% RSLogix 500 project Digital_Filling_Station.RSS, saved by version 8.30.00.16 %
PROJECT "P2"    % processor: Bul.1763 MicroLogix 1100 Series B %

PROGRAM FILES
  LAD 2   4 rungs
  LAD 3 "IO"  8 rungs
  LAD 4 "CONTROL"  6 rungs
  LAD 5 "CYCLE"  5 rungs

DATA FILES
  O0 OUTPUT  4 elements
  I1 INPUT  6 elements
  S2 STATUS  66 elements
  B3 BINARY  1 elements
  T4 TIMER  1 elements
  C5 COUNTER  1 elements
  R6 CONTROL  1 elements
  N7 INTEGER  1 elements
  F8 FLOAT  1 elements

LADDER 2
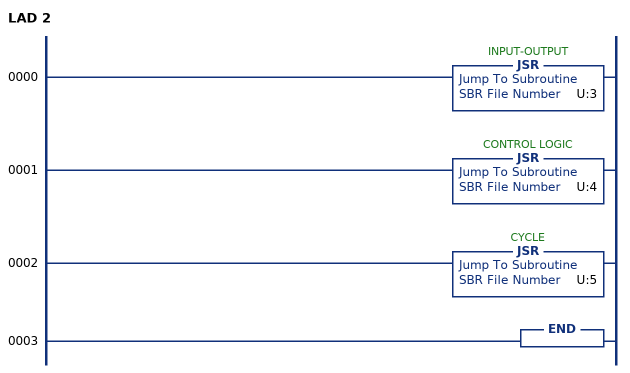
% Rung: 0 %
SOR JSR U:3 EOR
%   U:3  "INPUT-OUTPUT" %
% Rung: 1 %
SOR JSR U:4 EOR
%   U:4  "CONTROL LOGIC" %
% Rung: 2 %
SOR JSR U:5 EOR
%   U:5  "CYCLE" %
% Rung: 3 %
SOR END EOR

LADDER 3 "IO"
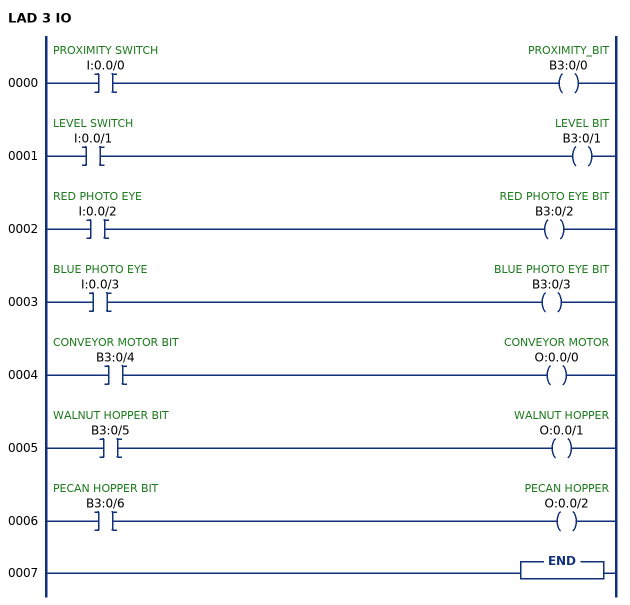
% Rung: 0 %
SOR XIC I:0.0/0 OTE B3:0/0 EOR
%   I:0.0/0  "PROXIMITY SWITCH" %
%   B3:0/0  "PROXIMITY_BIT" %
% Rung: 1 %
SOR XIC I:0.0/1 OTE B3:0/1 EOR
%   I:0.0/1  "LEVEL SWITCH" %
%   B3:0/1  "LEVEL BIT" %
% Rung: 2 %
SOR XIC I:0.0/2 OTE B3:0/2 EOR
%   I:0.0/2  "RED PHOTO EYE" %
%   B3:0/2  "RED PHOTO EYE BIT" %
% Rung: 3 %
SOR XIC I:0.0/3 OTE B3:0/3 EOR
%   I:0.0/3  "BLUE PHOTO EYE" %
%   B3:0/3  "BLUE PHOTO EYE BIT" %
% Rung: 4 %
SOR XIC B3:0/4 OTE O:0.0/0 EOR
%   B3:0/4  "CONVEYOR MOTOR BIT" %
%   O:0.0/0  "CONVEYOR MOTOR" %
% Rung: 5 %
SOR XIC B3:0/5 OTE O:0.0/1 EOR
%   B3:0/5  "WALNUT HOPPER BIT" %
%   O:0.0/1  "WALNUT HOPPER" %
% Rung: 6 %
SOR XIC B3:0/6 OTE O:0.0/2 EOR
%   B3:0/6  "PECAN HOPPER BIT" %
%   O:0.0/2  "PECAN HOPPER" %
% Rung: 7 %
SOR END EOR

LADDER 4 "CONTROL"
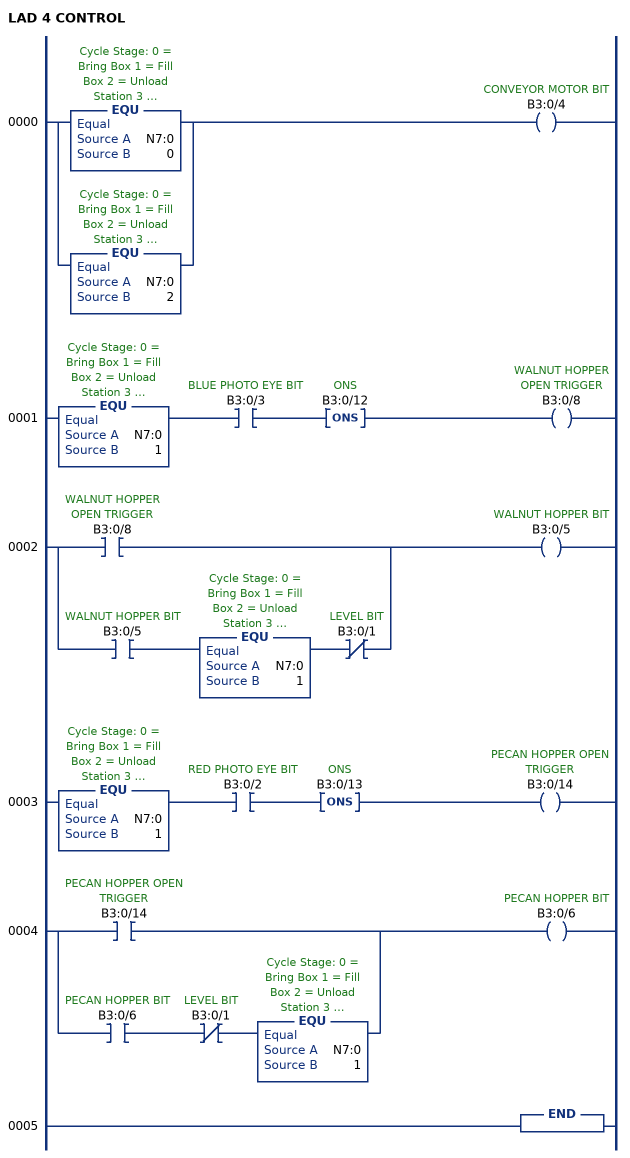
% Rung: 0 %
SOR BST EQU N7:0 0 NXB EQU N7:0 2 BND OTE B3:0/4 EOR
%   N7:0  "Cycle Stage: 0 = Bring Box 1 = Fill Box 2 = Unload Station 3 = Intermediate" %
%   B3:0/4  "CONVEYOR MOTOR BIT" %
% Rung: 1 %
SOR EQU N7:0 1 XIC B3:0/3 ONS B3:0/12 OTE B3:0/8 EOR
%   N7:0  "Cycle Stage: 0 = Bring Box 1 = Fill Box 2 = Unload Station 3 = Intermediate" %
%   B3:0/3  "BLUE PHOTO EYE BIT" %
%   B3:0/12  "ONS" %
%   B3:0/8  "WALNUT HOPPER OPEN TRIGGER" %
% Rung: 2 %
SOR BST XIC B3:0/8 NXB XIC B3:0/5 EQU N7:0 1 XIO B3:0/1 BND OTE B3:0/5 EOR
%   B3:0/8  "WALNUT HOPPER OPEN TRIGGER" %
%   B3:0/5  "WALNUT HOPPER BIT" %
%   N7:0  "Cycle Stage: 0 = Bring Box 1 = Fill Box 2 = Unload Station 3 = Intermediate" %
%   B3:0/1  "LEVEL BIT" %
% Rung: 3 %
SOR EQU N7:0 1 XIC B3:0/2 ONS B3:0/13 OTE B3:0/14 EOR
%   N7:0  "Cycle Stage: 0 = Bring Box 1 = Fill Box 2 = Unload Station 3 = Intermediate" %
%   B3:0/2  "RED PHOTO EYE BIT" %
%   B3:0/13  "ONS" %
%   B3:0/14  "PECAN HOPPER OPEN TRIGGER" %
% Rung: 4 %
SOR BST XIC B3:0/14 NXB XIC B3:0/6 XIO B3:0/1 EQU N7:0 1 BND OTE B3:0/6 EOR
%   B3:0/14  "PECAN HOPPER OPEN TRIGGER" %
%   B3:0/6  "PECAN HOPPER BIT" %
%   B3:0/1  "LEVEL BIT" %
%   N7:0  "Cycle Stage: 0 = Bring Box 1 = Fill Box 2 = Unload Station 3 = Intermediate" %
% Rung: 5 %
SOR END EOR

LADDER 5 "CYCLE"
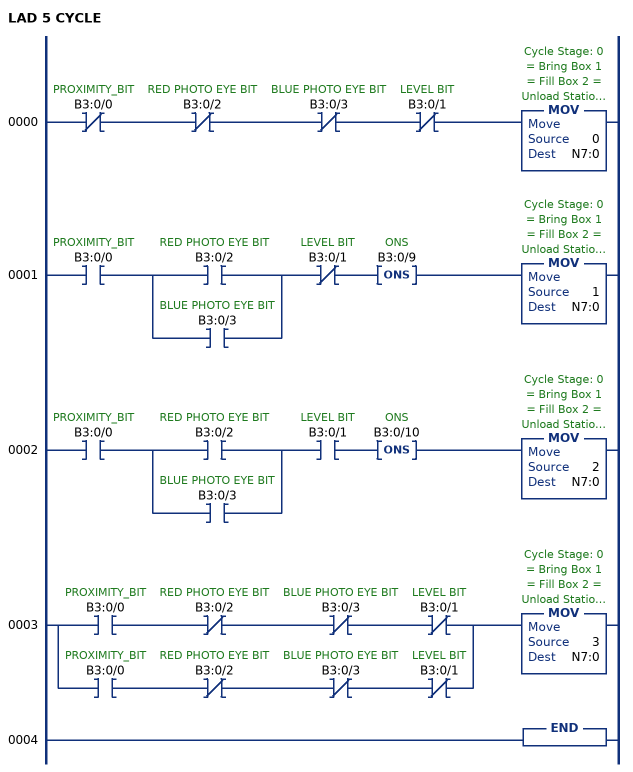
% Rung: 0 %
SOR XIO B3:0/0 XIO B3:0/2 XIO B3:0/3 XIO B3:0/1 MOV 0 N7:0 EOR
%   B3:0/0  "PROXIMITY_BIT" %
%   B3:0/2  "RED PHOTO EYE BIT" %
%   B3:0/3  "BLUE PHOTO EYE BIT" %
%   B3:0/1  "LEVEL BIT" %
%   N7:0  "Cycle Stage: 0 = Bring Box 1 = Fill Box 2 = Unload Station 3 = Intermediate" %
% Rung: 1 %
SOR XIC B3:0/0 BST XIC B3:0/2 NXB XIC B3:0/3 BND XIO B3:0/1 ONS B3:0/9 MOV 1 N7:0 EOR
%   B3:0/0  "PROXIMITY_BIT" %
%   B3:0/2  "RED PHOTO EYE BIT" %
%   B3:0/3  "BLUE PHOTO EYE BIT" %
%   B3:0/1  "LEVEL BIT" %
%   B3:0/9  "ONS" %
%   N7:0  "Cycle Stage: 0 = Bring Box 1 = Fill Box 2 = Unload Station 3 = Intermediate" %
% Rung: 2 %
SOR XIC B3:0/0 BST XIC B3:0/2 NXB XIC B3:0/3 BND XIC B3:0/1 ONS B3:0/10 MOV 2 N7:0 EOR
%   B3:0/0  "PROXIMITY_BIT" %
%   B3:0/2  "RED PHOTO EYE BIT" %
%   B3:0/3  "BLUE PHOTO EYE BIT" %
%   B3:0/1  "LEVEL BIT" %
%   B3:0/10  "ONS" %
%   N7:0  "Cycle Stage: 0 = Bring Box 1 = Fill Box 2 = Unload Station 3 = Intermediate" %
% Rung: 3 %
SOR BST XIC B3:0/0 XIO B3:0/2 XIO B3:0/3 XIO B3:0/1 NXB XIC B3:0/0 XIO B3:0/2 XIO B3:0/3 XIO B3:0/1 BND MOV 3 N7:0 EOR
%   B3:0/0  "PROXIMITY_BIT" %
%   B3:0/2  "RED PHOTO EYE BIT" %
%   B3:0/3  "BLUE PHOTO EYE BIT" %
%   B3:0/1  "LEVEL BIT" %
%   N7:0  "Cycle Stage: 0 = Bring Box 1 = Fill Box 2 = Unload Station 3 = Intermediate" %
% Rung: 4 %
SOR END EOR
